// TIA Portal project "eip" (V16)

(* hardware
DEVICE "S7-1200 station_1"  S7-1200 Station
   slot 0: "Rack_0"  S7-1200 Rack  Rack  V1.0
   slot 1: "PLC_L"  CPU 1214C AC/DC/Rly  6ES7 214-1BG40-0XB0  V4.4
   slot 2: "DI 8/DQ 8x24VDC_1"  6ES7 223-1BH32-0XB0  V2.0
DEVICE "S7-1200 station_2"  S7-1200 Station
   slot 0: "Rack_0"  S7-1200 Rack  Rack  V1.0
   slot 1: "PLC_R"  CPU 1214C AC/DC/Rly  6ES7 214-1BG40-0XB0  V4.4
   slot 2: "DI 8/DQ 8x24VDC_1"  6ES7 223-1BH32-0XB0  V2.0
   slot 3: "AI 4x13BIT/AQ 2x14BIT_1"  6ES7 234-4HE32-0XB0  V2.1
*)

// ===== PLC "PLC_L"  CPU 1214C AC/DC/Rly =====
// protected blocks, not shown: "LCCF_EnetScanner"

// folder: S7-1200/data types

TYPE "LCCF_typeDiagnostics"
TITLE = typeEtherNetIpDiagnostics
// Contains extendend diagnosis functions for debugging purposes.
   STRUCT
      status : Word := 16#7000;   // Status of the Block or error identification when error occurred
      subfunctionStatus : Word;   // Status or return value of called FB's, FCs and system blocks
      stateNumber : DInt;   // State in the Block when the error occurred
   END_STRUCT;
END_TYPE

TYPE "LCCF_typeEnetAdaptConfig"
TITLE = typeEtherNetIpAdapterConfig
// Contains required information about the EtherNet/IP adapter to communicate with
   STRUCT
      address : IP_V4;   // IP v4 address of the adapter to access
      vendorIdentifier : UInt;   // ODVA assigned Vendor ID (from EDS files)
      productType : UInt;   // ODVA assigned ProductType number (from EDS files)
      productCode : UInt;   // ODVA assigned ProductCode (from EDS files)
      revisionMajor : USInt;   // MajorRevision
      revisionMinor : USInt;   // MinorRevision
      assemblyInstance : UInt;   // Instance the Assembly can be reached at (from EDS file)
      packetInterval : Time;   // Requested Packet Interval/ Update Rate
      conPointOutputIdentifier : UInt;   // Connection Point Identifier O->T direction
      conPointOutputSize : UInt;   // [Bytes] Connection Point Size in Bytes O->T direction
      conPointInputIdentifier : UInt;   // Connection Point Identifier T->O direction
      conPointInputSize : UInt;   // [Bytes] Connection Point Size in Bytes O->T direction
      configDataSize : UInt;   // [Bytes] Configuration data size of the assembly instance
   END_STRUCT;
END_TYPE

TYPE "LCCF_typeEnetAdaptData"
TITLE = typeEnetAdptData
// Provides the data areas for each adapter in the maximum supported size
   STRUCT
      inputs : Array[0..501] of USInt;   // contains the input data sent from the adapter
      outputs : Array[0..497] of USInt;   // contains the output data sent to the adapter
      configs : Array[0..399] of USInt;   // contains configuration data for the adapter transmitted on startup
   END_STRUCT;
END_TYPE

// folder: (top level)

DATA_BLOCK "Data_block_1"   // DB2
{ S7_Optimized_Access := 'TRUE' }
VERSION : 0.1
   VAR
      adapters : Array[0..0] of "LCCF_typeEnetAdaptConfig";
      datas : Array[0..0] of "LCCF_typeEnetAdaptData";
   END_VAR
BEGIN
   adapters[0].address.ADDR[1] := 192;
   adapters[0].address.ADDR[2] := 168;
   adapters[0].vendorIdentifier := 1251;
   adapters[0].productType := 12;
   adapters[0].productCode := 1200;
   adapters[0].revisionMajor := 1;
   adapters[0].revisionMinor := 4;
   adapters[0].conPointOutputIdentifier := 102;
   adapters[0].conPointInputIdentifier := 101;
   adapters[0].packetInterval := T#10ms;
   adapters[0].conPointOutputSize := 1;
   adapters[0].conPointInputSize := 1;
   adapters[0].assemblyInstance := 104;
   adapters[0].address.ADDR[3] := 0;
   adapters[0].address.ADDR[4] := 102;
   adapters[0].configDataSize := 1;
END_DATA_BLOCK

ORGANIZATION_BLOCK "Main"   // OB1, LAD, ProgramCycle
TITLE = "Main Program Sweep (Cycle)"
{ S7_Optimized_Access := 'TRUE' }
VERSION : 0.1
   VAR_INPUT
      Initial_Call : Bool;   // Initial call of this OB
      Remanence : Bool;   // =True, if remanent data are available
   END_VAR
BEGIN

REGION Network 1
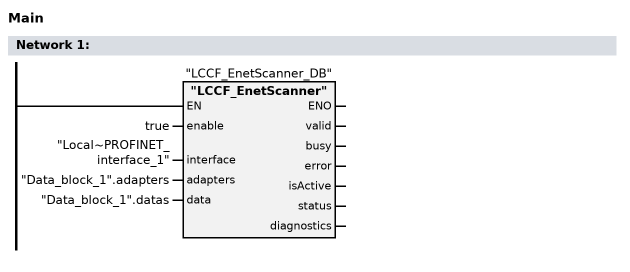
   RUNG wire#powerrail
      "LCCF_EnetScanner_DB"(enable := true, interface := "Local~PROFINET_interface_1", adapters := "Data_block_1".adapters, data := "Data_block_1".datas, valid =>, busy =>, error =>, isActive =>, status =>, diagnostics =>)
   END_RUNG
   // the same network as SCL:
   "LCCF_EnetScanner_DB"(enable := true,   // "LCCF_EnetScanner"
                         interface := "Local~PROFINET_interface_1",
                         adapters := "Data_block_1".adapters,
                         data := "Data_block_1".datas);
END_REGION
END_ORGANIZATION_BLOCK

ORGANIZATION_BLOCK "Main_1"   // OB123, SCL, ProgramCycle
TITLE = "Main Program Sweep (Cycle)"
{ S7_Optimized_Access := 'TRUE' }
VERSION : 0.1
   VAR_INPUT
      Initial_Call : Bool;   // Initial call of this OB
      Remanence : Bool;   // =True, if remanent data are available
   END_VAR
   VAR_TEMP
      t : Int;
   END_VAR
   VAR CONSTANT
      "b" : Int;
   END_VAR
BEGIN
   "Data_block_1".datas[0].outputs[1] := "Data_block_1".datas[0].outputs[1] + 1;
   IF "Data_block_1".datas[0].outputs[1] = 10 THEN
       "Data_block_1".datas[0].outputs[0] := "Data_block_1".datas[0].outputs[0] + 1;
       "Data_block_1".datas[0].outputs[1] := 0;
   END_IF;
   IF "Data_block_1".datas[0].outputs[0] >= 1000 THEN
       "Data_block_1".datas[0].outputs[0] := 0;
   END_IF;
END_ORGANIZATION_BLOCK

// ===== PLC "PLC_R"  CPU 1214C AC/DC/Rly =====
// protected blocks, not shown: "LCCF_EnetAdapter"

// folder: S7-1200/data types

TYPE "LCCF_typeAdaptDiag"
TITLE = typeAdaptDiag
// Contains extendend diagnosis functions for debugging purposes.
   STRUCT
      status : Word := 16#7000;   // Status of the Block or error identification when error occurred
      subfunctionStatus : Word;   // Status or return value of called FB's, FCs and system blocks
      stateNumber : DInt;   // State in the Block when the error occurred
      connectionIndex : DInt;   // Index to the connection causing the error
      subStateNumber : DInt;   // State of the Sub State Machine when the error occured
   END_STRUCT;
END_TYPE

// folder: (top level)

DATA_BLOCK "Data_block_1"   // DB2
{ S7_Optimized_Access := 'TRUE' }
VERSION : 0.1
   VAR
      inputs : Array[0..497] of SInt;
      outputs : Array[0..501] of SInt;
      config : Array[0..399] of SInt;
   END_VAR
BEGIN
   inputs[0] := 0;
END_DATA_BLOCK

ORGANIZATION_BLOCK "Main"   // OB1, LAD, ProgramCycle
TITLE = "Main Program Sweep (Cycle)"
{ S7_Optimized_Access := 'TRUE' }
VERSION : 0.1
   VAR_INPUT
      Initial_Call : Bool;   // Initial call of this OB
      Remanence : Bool;   // =True, if remanent data are available
   END_VAR
BEGIN

REGION Network 1
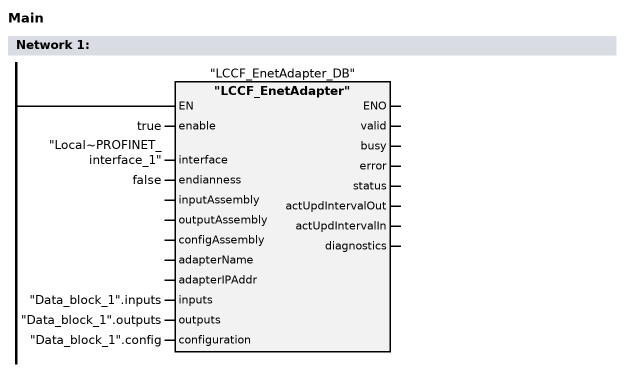
   RUNG wire#powerrail
      "LCCF_EnetAdapter_DB"(enable := true, interface := "Local~PROFINET_interface_1", endianness := false, inputAssembly :=, outputAssembly :=, configAssembly :=, adapterName :=, adapterIPAddr :=, inputs := "Data_block_1".inputs, outputs := "Data_block_1".outputs, configuration := "Data_block_1".config, valid =>, busy =>, error =>, status =>, actUpdIntervalOut =>, actUpdIntervalIn =>, diagnostics =>)
   END_RUNG
   // the same network as SCL:
   "LCCF_EnetAdapter_DB"(enable := true,   // "LCCF_EnetAdapter"
                         interface := "Local~PROFINET_interface_1",
                         endianness := false,
                         inputs := "Data_block_1".inputs,
                         outputs := "Data_block_1".outputs,
                         configuration := "Data_block_1".config);
END_REGION
END_ORGANIZATION_BLOCK